// This function has been automatically generated from the project information.
{attribute 'signature_flag' := '1073741824'}
{attribute 'TcGenerated'}
{attribute 'no-analysis'}
FUNCTION F_GetCompany : WSTRING
VAR_INPUT
	
END_VAR

F_GetCompany := "Course_OOP";

END_FUNCTION

(* stored: Version 1.1.0.1
   POU F_GetCompany: Id {6a927c5c-ed4a-0468-0986-1a3737a00842}, SpecialFunc None *)
